// TwinCAT 3 PLC project RecipeManagementSample
// ProgramVersion: 3.1.4022.0
// libraries:
//   Tc2_Standard, * (Beckhoff Automation GmbH)
//   Tc2_System, * (Beckhoff Automation GmbH)
//   Tc3_Module, * (Beckhoff Automation GmbH)
//   VisuDialogs, * (System)
// project tree:
//   / GlobalTextList.TcGTLO, PlcTask.TcTTO, RecipeManager.TcRMO (not stored), VisualizationManager.TcVMO (not stored), VISU_TASK.TcTTO
//   GVLs/ GVL_RecipeTable.TcGVL
//   POUs/ MAIN.TcPOU, RecipeManagement.TcPOU
//   VISUs/ Visualization.TcVIS
// real-time tasks:
//   TASK PlcTask: cycle T#10ms, priority 20, ADS port 350
//   TASK VISU_TASK: cycle T#200000us, priority 30, ADS port 351

CONFIGURATION RecipeManagementSample
    RESOURCE PLC ON TwinCAT3
        TASK PlcTask(INTERVAL := T#10ms, PRIORITY := 20);
        TASK VISU_TASK(INTERVAL := T#200000us, PRIORITY := 30);
        PROGRAM MAIN WITH PlcTask : MAIN;
        PROGRAM VisuElems_Visu_Prg WITH VISU_TASK : VisuElems.Visu_Prg;
        PROGRAM RecipeManagement WITH VISU_TASK : RecipeManagement;
    END_RESOURCE
END_CONFIGURATION

// ---- GVLs/GVL_RecipeTable.TcGVL
VAR_GLOBAL
	aRecipeNames 			: ARRAY[0..cMaxTableRows] OF STRING;
	aVariableNames 			: ARRAY[0..cMaxTableRows] OF STRING;
	aVariableValues 		: ARRAY[0..cMaxTableRows] OF STRING;
	nVariableIndex			: INT;
	nVariableCount 			: INT;
	nRecipeIndex 			: INT;
	nRecipeSelectionIndex 	: INT := -1;
	nRecipeCount 			: INT;
END_VAR
VAR_GLOBAL CONSTANT
	cMaxTableRows 			: INT := 9;
END_VAR

// ---- POUs/MAIN.TcPOU
PROGRAM MAIN
VAR
	nValueInt 	: INT;
	nValueDword : DWORD;
	fValueReal 	: REAL;
	
	sRecipe 	: STRING;
END_VAR

END_PROGRAM

// ---- POUs/RecipeManagement.TcPOU
PROGRAM RecipeManagement
VAR
	fbRecipeManCommands 	: RecipeManCommands; (* Recipe Manager *)
	
	bInit 					: BOOL := TRUE;
	
	nLastError 				: DWORD; (* Error from Recipe Manager *)
	nRecipeCount 			: INT;
	
	sRecipeDef 				: STRING := 'RecipeDefinition1'; (* current recipe definition *)
	sRecipe 				: STRING; (*Selected recipe *)
	nPreviousIndex			: INT; (* Previous selected index *)
	nPreviousSelectionIndex	: INT := -1; (* *)
	bReload 				: BOOL; (* Refresh recipes from files *)
	fbSaveVariablesTrigger	: R_TRIG;
	bSaveVariables			: BOOL;
	nSelectionIndexInList 	: INT;
	nCount					: INT;
	bReloadValues			: BOOL;
END_VAR

(* Initialization *)
IF bInit THEN
	(* Save the number of recipes in the specified recipe definition in a globar variable.*)
	GVL_RecipeTable.nRecipeCount := fbRecipeManCommands.GetRecipeCount(sRecipeDef);
	
	(* Empty all arrays *)
	FOR nCount := 0 TO cMaxTableRows DO
		GVL_RecipeTable.aRecipeNames[nCount] := '';
		GVL_RecipeTable.aVariableNames[nCount] := '';
		GVL_RecipeTable.aVariableValues[nCount] := '';
	END_FOR
	
	(* save all recipe names of the default recipe definition in an array *)
	fbRecipeManCommands.GetRecipeNames(	sRecipeDef,
										ADR(GVL_RecipeTable.aRecipeNames),
										10,
										GVL_RecipeTable.nRecipeIndex);
										
	GVL_RecipeTable.nRecipeSelectionIndex := -1;
	nPreviousSelectionIndex := -1;
	
	bInit := FALSE;
END_IF

(* Count all recipes in the defined recipe definition *)
nRecipeCount := fbRecipeManCommands.GetRecipeCount(sRecipeDef);
nLastError := fbRecipeManCommands.GetLastError();

(* Scroll position of the recipe list has changed. *)
IF GVL_RecipeTable.nRecipeIndex <> nPreviousIndex THEN
	fbRecipeManCommands.GetRecipeNames(	sRecipeDef,
										ADR(GVL_RecipeTable.aRecipeNames),
										10,
										GVL_RecipeTable.nRecipeIndex);
	nPreviousIndex := GVL_RecipeTable.nRecipeIndex;
END_IF

(* Selection of the current recipe has changed *)
IF GVL_RecipeTable.nRecipeSelectionIndex <> nPreviousSelectionIndex OR bReloadValues THEN
	nPreviousSelectionIndex := GVL_RecipeTable.nRecipeSelectionIndex;
	nSelectionIndexInList := GVL_RecipeTable.nRecipeSelectionIndex - GVL_RecipeTable.nRecipeIndex;
	
	(* Get the selected recipe name *)
	IF nSelectionIndexInList >= 0 AND nSelectionIndexInList < 10 THEN
		sRecipe := GVL_RecipeTable.aRecipeNames[nSelectionIndexInList];
	END_IF
	
	fbRecipeManCommands.GetRecipeValues(sRecipeDef,
										sRecipe,
										ADR(GVL_RecipeTable.aVariableValues),
										10,
										GVL_RecipeTable.nVariableIndex,
										80);
										
	fbRecipeManCommands.GetRecipeVariableNames(	sRecipeDef,
												sRecipe,
												ADR(GVL_RecipeTable.aVariableNames),
												10,
												GVL_RecipeTable.nVariableIndex);
	
	bReloadValues := FALSE;
END_IF

(* Reload the recipe list from the file system *)
IF bReload THEN
	fbRecipeManCommands.ReloadRecipes(sRecipeDef);
	bInit := TRUE;
	bReload := FALSE;
END_IF

(* Save the edited values into the recipe *)
fbSaveVariablesTrigger(CLK := bSaveVariables);
IF fbSaveVariablesTrigger.Q THEN
	fbRecipeManCommands.SetRecipeValues(sRecipeDef,
										sRecipe,
										ADR(GVL_RecipeTable.aVariableValues),
										10,
										GVL_RecipeTable.nVariableIndex);	
	bSaveVariables := FALSE;
END_IF

END_PROGRAM

// ---- GlobalTextList.TcGTLO
TEXTLIST GlobalTextList
  680 = '%s'
  233 = 'All recipe values crom the current recipe are listed in this table.\nPressing the "Save" button will set the current values in the recipe. Pressing "Save Recipe" afterwards will save the recipe in a file.'
  232 = 'All recipes from the current recipe definition are listed in this table.\nPressing the "Refresh" button will reload all recipe files.'
  676 = 'Create Recipe'
  33 = 'Create recipe'
  3 = 'Current PLC values'
  236 = 'Current Recipe Definiton:'
  938 = 'Current recipe definiton:'
  60 = 'Current Recipe:'
  668 = 'Current recipe:'
  311 = 'Current Recipe: %s'
  621 = 'Current Values'
  231 = 'Delete Recipe'
  895 = 'Delete recipe'
  1 = 'DWORD value:'
  737 = 'GroupBox'
  0 = 'INT value:'
  61 = 'Last Error (0 == OK):'
  992 = 'Last error (0 == OK):'
  670 = 'Last Error 0 == OK: %s'
  976 = 'List of available recipes for the current recipe definiton'
  7 = 'List of available recipes for the current recipe definiton:'
  900 = 'List of existing recipes for the current recipe definiton:'
  675 = 'Load Recipe'
  897 = 'Load recipe'
  229 = 'Load Recipe From'
  918 = 'Load recipe from'
  226 = 'Name'
  4 = "Name and value of the current recipe's variables:"
  230 = 'Name and Value of the Current Recipe:'
  709 = 'Name and value of the current recipe:'
  79 = 'New recipe name:'
  63 = 'New Recipe Name:'
  679 = 'New Recipe Name: \n%s'
  673 = 'Read Variables into Recipe'
  722 = 'Read variables into recipe'
  514 = 'Read variables into Recipe'
  2 = 'REAL value:'
  365 = 'Recipe commands'
  62 = 'Recipe Count:'
  15 = 'Recipe count:'
  671 = 'Recipe Count: %s'
  234 = 'Recipe Execute Commands:'
  740 = 'Recipe information'
  407 = 'Recipe Management'
  225 = 'Recipes'
  865 = 'Refresh'
  224 = 'Save'
  674 = 'Save Recipe'
  327 = 'Save recipe'
  228 = 'Save Recipe As'
  272 = 'Save recipe as'
  866 = 'SelectionIndex: %s'
  227 = 'Value'
  877 = 'Value 1:'
  672 = 'Value 1: %s'
  181 = 'Value 2:'
  677 = 'Value 2: %s'
  921 = 'Value 3:'
  235 = 'Value 3: %s'
  969 = 'Values'
  678 = 'Write Recipe into Variables'
  244 = 'Write recipe into variables'
END_TEXTLIST

// ---- VISUs/Visualization.TcVIS
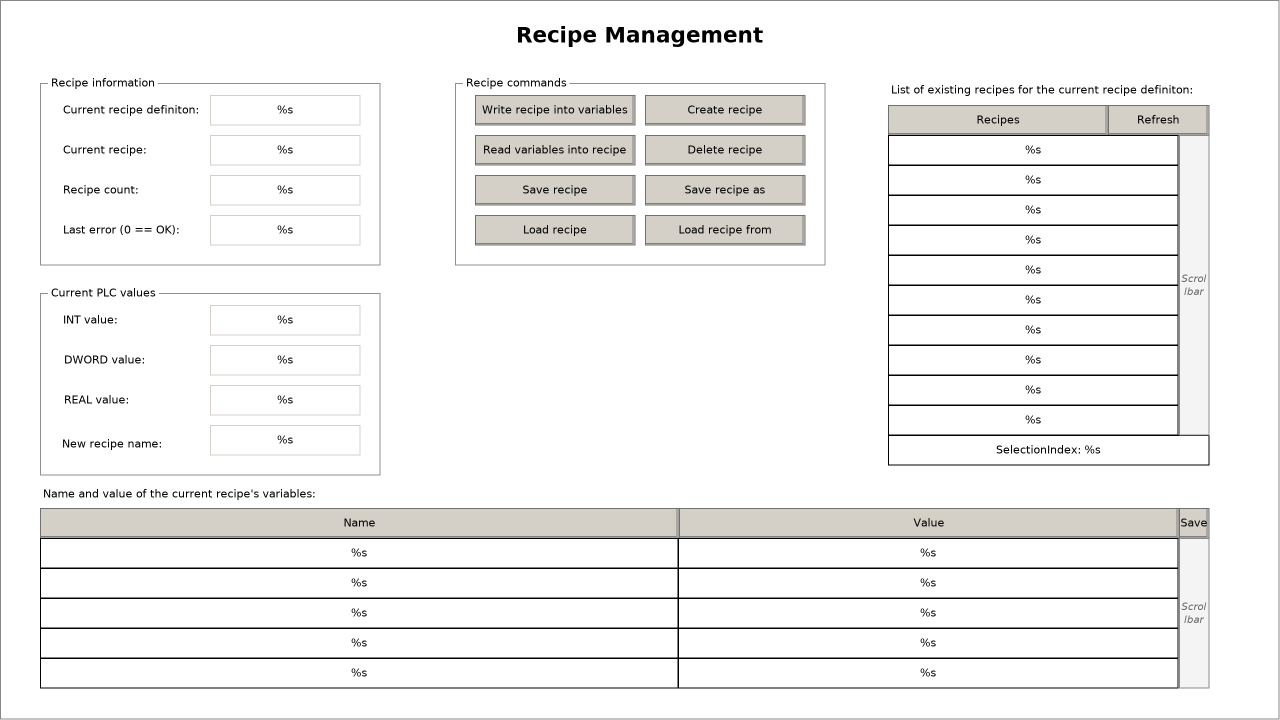
VISUALIZATION Visualization  // 1280x720
    GroupBox (455,75 370x190), "Recipe commands"
        Button (20,20 160x30), "Write recipe into variables"
            OnMouseClick: ExecuteCommand ExecuteCommand=ExecuteCommand=[Command=WriteRecipe, Value=RecipeManagement.sRecipeDef, Value2=RecipeManagement.sRecipe]
        Button (20,60 160x30), "Read variables into recipe"
            OnMouseClick: ExecuteCommand ExecuteCommand=ExecuteCommand=[Command=ReadRecipe, Value=RecipeManagement.sRecipeDef, Value2=RecipeManagement.sRecipe]
            OnMouseClick: execute { RecipeManagement.bReloadValues := TRUE; }
        Button (20,100 160x30), "Save recipe"
            OnMouseClick: ExecuteCommand ExecuteCommand=ExecuteCommand=[Command=SaveRecipe, Value=RecipeManagement.sRecipeDef, Value2=RecipeManagement.sRecipe]
        Button (20,140 160x30), "Load recipe"
            OnMouseClick: ExecuteCommand ExecuteCommand=ExecuteCommand=[Command=LoadRecipe, Value=RecipeManagement.sRecipeDef, Value2=RecipeManagement.sRecipe]
            OnMouseClick: toggle RecipeManagement.bReloadValues
        Button (190,20 160x30), "Create recipe"
            OnMouseClick: ExecuteCommand ExecuteCommand=ExecuteCommand=[Command=CreateRecipe, Value=RecipeManagement.sRecipeDef, Value2=MAIN.sRecipe]
            OnMouseClick: execute { RecipeManagement.bReload := TRUE; }
        Button (190,100 160x30), "Save recipe as"
            OnMouseClick: ExecuteCommand ExecuteCommand=ExecuteCommand=[Command=SaveRecipeAs, Value=RecipeManagement.sRecipeDef, Value2=RecipeManagement.sRecipe]
        Button (190,140 160x30), "Load recipe from"
            OnMouseClick: ExecuteCommand ExecuteCommand=ExecuteCommand=[Command=LoadRecipeFrom, Value=RecipeManagement.sRecipeDef, Value2=RecipeManagement.sRecipe]
        Button (190,60 160x30), "Delete recipe"
            OnMouseClick: ExecuteCommand ExecuteCommand=ExecuteCommand=[Command=DeleteRecipe, Value=RecipeManagement.sRecipeDef, Value2=RecipeManagement.sRecipe]
            OnMouseClick: execute { RecipeManagement.bInit := TRUE; }
    GroupBox (40,285 340x190), "Current PLC values"
        Label (20,20 150x30), "INT value:"
        Textfield (170,20 150x30), "%s", text variable: MAIN.nValueInt
            OnMouseClick: write the text variable via Default
        Label (21,60 150x30), "DWORD value:"
        Textfield (170,60 150x30), "%s", text variable: MAIN.nValueDword
            OnMouseClick: write the text variable via Default
        Label (21,100 150x30), "REAL value:"
        Textfield (170,100 150x30), "%s", text variable: MAIN.fValueReal
            OnMouseClick: write the text variable via Default
        Label (19,144 150x30), "New recipe name:"
        Textfield (170,140 150x30), "%s", text variable: MAIN.sRecipe
            OnMouseClick: write the text variable via Default
    Label (490,20 300x30), "Recipe Management"
    GroupBox (40,75 340x190), "Recipe information"
        Textfield (170,20 150x30), "%s", text variable: RecipeManagement.sRecipeDef
            OnMouseClick: write the text variable via Default
        Label (20,20 150x30), "Current recipe definiton:"
        Label (20,60 150x30), "Current recipe:"
        Label (20,140 150x30), "Last error (0 == OK):"
        Label (20,100 150x30), "Recipe count:"
        Textfield (170,60 150x30), "%s", text variable: RecipeManagement.sRecipe
            OnMouseClick: write the text variable via Default
        Textfield (170,140 150x30), "%s", text variable: RecipeManagement.nLastError
        Textfield (170,100 150x30), "%s", text variable: RecipeManagement.nRecipeCount
    Button (40,508 639x30), "Name"
        OnMouseDown: toggle RecipeManagement.bReload
    Button (679,508 500x30), "Value"
        OnMouseDown: toggle RecipeManagement.bReload
    Rectangle (40,479 305x30), "Name and value of the current recipe's variables:"
    Button (1179,508 30x30), "Save"
        OnMouseDown: toggle RecipeManagement.bSaveVariables
    Rectangle (40,538 638x30), "%s", text variable: GVL_RecipeTable.aVariableNames[0]
    Rectangle (40,568 638x30), "%s", text variable: GVL_RecipeTable.aVariableNames[1]
    Rectangle (40,598 638x30), "%s", text variable: GVL_RecipeTable.aVariableNames[2]
    Rectangle (40,628 638x30), "%s", text variable: GVL_RecipeTable.aVariableNames[3]
    Rectangle (40,658 638x30), "%s", text variable: GVL_RecipeTable.aVariableNames[4]
    Rectangle (678,538 500x30), "%s", text variable: GVL_RecipeTable.aVariableValues[0]
        OnMouseDown: write the text variable via Edit
    Rectangle (678,568 500x30), "%s", text variable: GVL_RecipeTable.aVariableValues[1]
        OnMouseDown: write the text variable via Edit
    Rectangle (678,598 500x30), "%s", text variable: GVL_RecipeTable.aVariableValues[2]
        OnMouseDown: write the text variable via Edit
    Rectangle (678,628 500x30), "%s", text variable: GVL_RecipeTable.aVariableValues[3]
        OnMouseDown: write the text variable via Edit
    Rectangle (678,658 500x30), "%s", text variable: GVL_RecipeTable.aVariableValues[4]
        OnMouseDown: write the text variable via Edit
    Scrollbar (1179,538 30x150)
        p2245068023: GVL_RecipeTable.nRecipeCount
        p1057716461: GVL_RecipeTable.nVariableIndex
    Button (888,105 220x30), "Recipes"
        OnMouseDown: toggle RecipeManagement.bReload
    Label (888,75 322x30), "List of existing recipes for the current recipe definiton:"
    Button (1108,105 101x30), "Refresh"
        OnMouseDown: toggle RecipeManagement.bReload
    Rectangle (888,135 290x30), "%s", text variable: GVL_RecipeTable.aRecipeNames[0], colour toggle: (GVL_RecipeTable.nRecipeSelectionIndex-GVL_RecipeTable.nRecipeIndex) = 0
        OnMouseDown: execute { GVL_RecipeTable.nRecipeSelectionIndex := GVL_RecipeTable.nRecipeIndex; }
    Rectangle (888,165 290x30), "%s", text variable: GVL_RecipeTable.aRecipeNames[1], colour toggle: (GVL_RecipeTable.nRecipeSelectionIndex-GVL_RecipeTable.nRecipeIndex) = 1
        OnMouseDown: execute { GVL_RecipeTable.nRecipeSelectionIndex := GVL_RecipeTable.nRecipeIndex + 1; }
    Rectangle (888,195 290x30), "%s", text variable: GVL_RecipeTable.aRecipeNames[2], colour toggle: (GVL_RecipeTable.nRecipeSelectionIndex-GVL_RecipeTable.nRecipeIndex) = 2
        OnMouseDown: execute { GVL_RecipeTable.nRecipeSelectionIndex := GVL_RecipeTable.nRecipeIndex + 2; }
    Rectangle (888,225 290x30), "%s", text variable: GVL_RecipeTable.aRecipeNames[4], colour toggle: (GVL_RecipeTable.nRecipeSelectionIndex-GVL_RecipeTable.nRecipeIndex) = 3
        OnMouseDown: execute { GVL_RecipeTable.nRecipeSelectionIndex := GVL_RecipeTable.nRecipeIndex + 3; }
    Rectangle (888,255 290x30), "%s", text variable: GVL_RecipeTable.aRecipeNames[5], colour toggle: (GVL_RecipeTable.nRecipeSelectionIndex-GVL_RecipeTable.nRecipeIndex) = 4
        OnMouseDown: execute { GVL_RecipeTable.nRecipeSelectionIndex := GVL_RecipeTable.nRecipeIndex + 4; }
    Rectangle (888,285 290x30), "%s", text variable: GVL_RecipeTable.aRecipeNames[6], colour toggle: (GVL_RecipeTable.nRecipeSelectionIndex-GVL_RecipeTable.nRecipeIndex) = 5
        OnMouseDown: execute { GVL_RecipeTable.nRecipeSelectionIndex := GVL_RecipeTable.nRecipeIndex + 5; }
    Rectangle (888,315 290x30), "%s", text variable: GVL_RecipeTable.aRecipeNames[6], colour toggle: (GVL_RecipeTable.nRecipeSelectionIndex-GVL_RecipeTable.nRecipeIndex) = 6
        OnMouseDown: execute { GVL_RecipeTable.nRecipeSelectionIndex := GVL_RecipeTable.nRecipeIndex + 6; }
    Rectangle (888,345 290x30), "%s", text variable: GVL_RecipeTable.aRecipeNames[7], colour toggle: (GVL_RecipeTable.nRecipeSelectionIndex-GVL_RecipeTable.nRecipeIndex) = 7
        OnMouseDown: execute { GVL_RecipeTable.nRecipeSelectionIndex := GVL_RecipeTable.nRecipeIndex + 7; }
    Rectangle (888,375 290x30), "%s", text variable: GVL_RecipeTable.aRecipeNames[8], colour toggle: (GVL_RecipeTable.nRecipeSelectionIndex-GVL_RecipeTable.nRecipeIndex) = 8
        OnMouseDown: execute { GVL_RecipeTable.nRecipeSelectionIndex := GVL_RecipeTable.nRecipeIndex + 8; }
    Rectangle (888,405 290x30), "%s", text variable: GVL_RecipeTable.aRecipeNames[9], colour toggle: (GVL_RecipeTable.nRecipeSelectionIndex-GVL_RecipeTable.nRecipeIndex) = 9
        OnMouseDown: execute { GVL_RecipeTable.nRecipeSelectionIndex := GVL_RecipeTable.nRecipeIndex + 9; }
    Rectangle (888,435 321x30), "SelectionIndex: %s", text variable: GVL_RecipeTable.nRecipeSelectionIndex+1
    Scrollbar (1179,135 30x300)
        p2245068023: GVL_RecipeTable.nRecipeCount
        p1057716461: GVL_RecipeTable.nRecipeIndex
END_VISUALIZATION
